(* Logix 5000 project; controller TEC_81 vendor 1 type 14 code 148 rev 36.11; software revision 36.00; part 5 of 5 *)
(* tags used below, declared in another part *)
   Lasers_OK : BOOL;   // Laser Scanner Close Loop Indicator
   LS_1 : DCI_STOP;   // Status of Laser Scanner 1
   LS_1_Status : BOOL;   // General status of inputs
   LS_2 : DCI_STOP;   // Status of Laser Scanner 2
   LS_2_Status : BOOL;   // General status of inputs
   Mat_1_Status : BOOL;   // General status of inputs
   ONS_Laser_1 : BOOL;   // One time execution for reset
   ONS_Laser_2 : BOOL;   // One time execution for reset
   Output_Enable_Laser_1 : BOOL;   // General status of Laser 1
   Output_Enable_Laser_2 : BOOL;   // General status of Laser 2
   Safety_Close_Loop_ok : BOOL;   // General Safety Indicator
   Safety_Mat_ok : BOOL;   // Safety Mat Close Loop Indicator
   Safety_Reset_General : BOOL;   // Unified General Reset
   AbrirInterlock_conveyor_Safety : BOOL;   // Mapped green button for interlock 2 opening
   AbrirInterlock_Principal_Safety : BOOL;   // Mapped green button for interlock 1 opening
   EStops_OK : BOOL;   // E-Stop Close Loop Indicator
   Interlocks_Ok : BOOL;   // Interlocks Close Loop Indicator
   LigthCurtain_ok : BOOL;   // Light Curtains Close Loop Indicator
   MC_1_Interlock : DCI_STOP;   // Status of Interlock 1
   MC_1_Interlock_Status : BOOL;   // General status of inputs
   MC_1_LigthCurtain : DCI_STOP;   // Status of Light Curtain 1
   MC_1_LigthCurtain_Status : BOOL;   // General status of inputs
   MC_2_Interlock : DCI_STOP;   // Status of Interlock 2
   MC_2_Interlock_Status : BOOL;   // General status of inputs
   MC_2_LightCurtain_Status : BOOL;   // General status of inputs
   MC_2_LigthCurtain : DCI_STOP;   // Status of Light Curtain 2
   Ons : INT;
   Operation_Mode : BOOL;   // Operation Mode for HMI (1) Manual (0) Automatico
   Reset_Almacen_1_Sfty : BOOL;
   Reset_Almacen_2_Sfty : BOOL;
   Reset_Principal_Sfty : BOOL;
   Reset_Salida_1_Sfty : BOOL;
   SafetyReset_almacen_1 : BOOL;   // Reset status Almacen 1
   SafetyReset_almacen_2 : BOOL;   // Reset status Almacen 2
   SafetyReset_Principal : BOOL;   // Reset status salida principal
   SafetyReset_Salida_1 : BOOL;   // Reset status Salida 1
   Storage_2 : BOOL;
   Storage_3 : BOOL;
   Storage_4 : BOOL;
   Storage_5 : BOOL;
(* SafetyProgram, continued *)

ROUTINE Interlocks   (* ladder *)
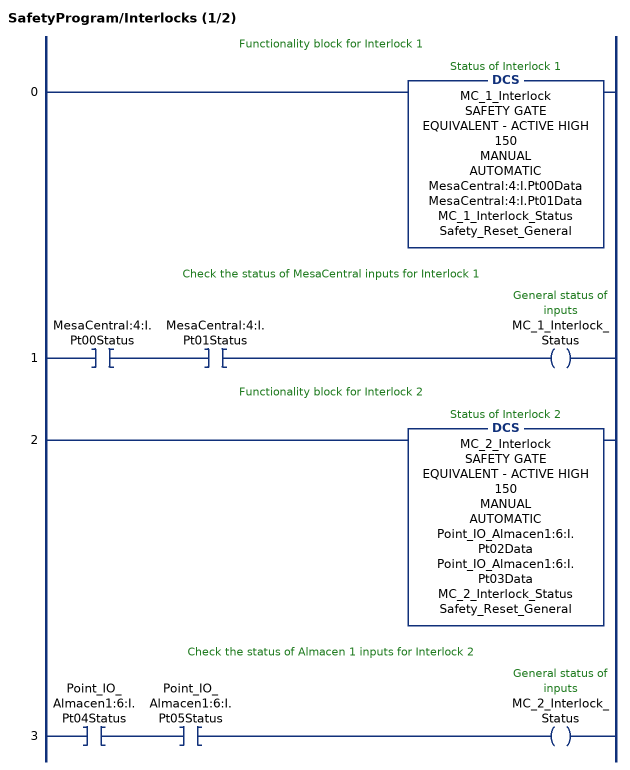
   // Functionality block for Interlock 1
   0: DCS(MC_1_Interlock,SAFETY GATE,EQUIVALENT - ACTIVE HIGH,150,MANUAL,AUTOMATIC,MesaCentral:4:I.Pt00Data,MesaCentral:4:I.Pt01Data,MC_1_Interlock_Status,Safety_Reset_General);
   // Check the status of MesaCentral inputs for Interlock 1
   1: XIC(MesaCentral:4:I.Pt00Status)XIC(MesaCentral:4:I.Pt01Status)OTE(MC_1_Interlock_Status);
   // Functionality block for Interlock 2
   2: DCS(MC_2_Interlock,SAFETY GATE,EQUIVALENT - ACTIVE HIGH,150,MANUAL,AUTOMATIC,Point_IO_Almacen1:6:I.Pt02Data,Point_IO_Almacen1:6:I.Pt03Data,MC_2_Interlock_Status,Safety_Reset_General);
   // Check the status of Almacen 1 inputs for Interlock 2
   3: XIC(Point_IO_Almacen1:6:I.Pt04Status)XIC(Point_IO_Almacen1:6:I.Pt05Status)OTE(MC_2_Interlock_Status);
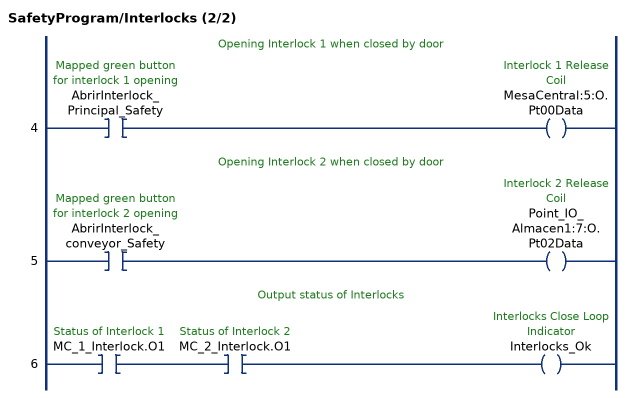
   // Opening Interlock 1 when closed by door
   4: XIC(AbrirInterlock_Principal_Safety)OTE(MesaCentral:5:O.Pt00Data);
   // Opening Interlock 2 when closed by door
   5: XIC(AbrirInterlock_conveyor_Safety)OTE(Point_IO_Almacen1:7:O.Pt02Data);
   // Output status of Interlocks
   6: XIC(MC_1_Interlock.O1)XIC(MC_2_Interlock.O1)OTE(Interlocks_Ok);
END_ROUTINE

ROUTINE Laser_Scanner   (* ladder *)
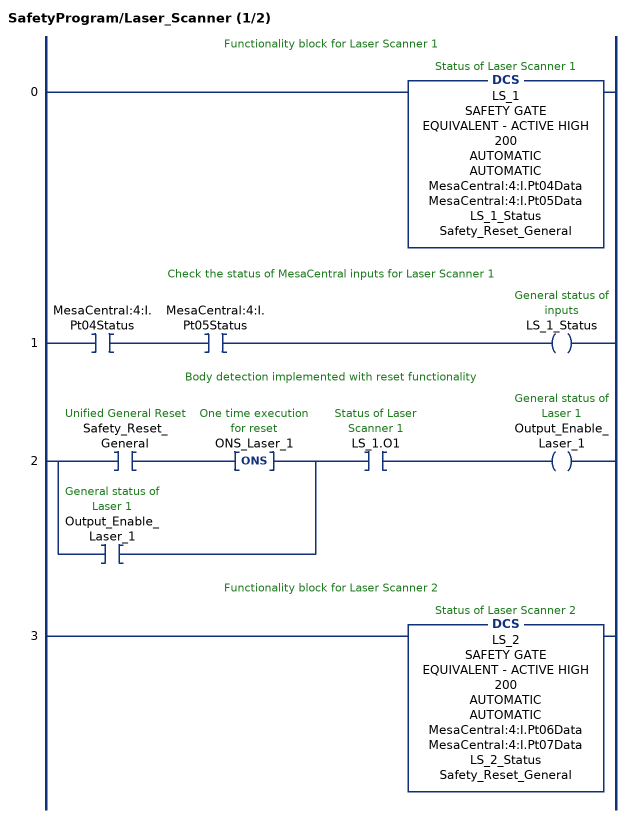
   // Functionality block for Laser Scanner 1
   0: DCS(LS_1,SAFETY GATE,EQUIVALENT - ACTIVE HIGH,200,AUTOMATIC,AUTOMATIC,MesaCentral:4:I.Pt04Data,MesaCentral:4:I.Pt05Data,LS_1_Status,Safety_Reset_General);
   // Check the status of MesaCentral inputs for Laser Scanner 1
   1: XIC(MesaCentral:4:I.Pt04Status)XIC(MesaCentral:4:I.Pt05Status)OTE(LS_1_Status);
   // Body detection implemented with reset functionality
   2: [XIC(Safety_Reset_General) ONS(ONS_Laser_1) ,XIC(Output_Enable_Laser_1) ]XIC(LS_1.O1)OTE(Output_Enable_Laser_1);
   // Functionality block for Laser Scanner 2
   3: DCS(LS_2,SAFETY GATE,EQUIVALENT - ACTIVE HIGH,200,AUTOMATIC,AUTOMATIC,MesaCentral:4:I.Pt06Data,MesaCentral:4:I.Pt07Data,LS_2_Status,Safety_Reset_General);
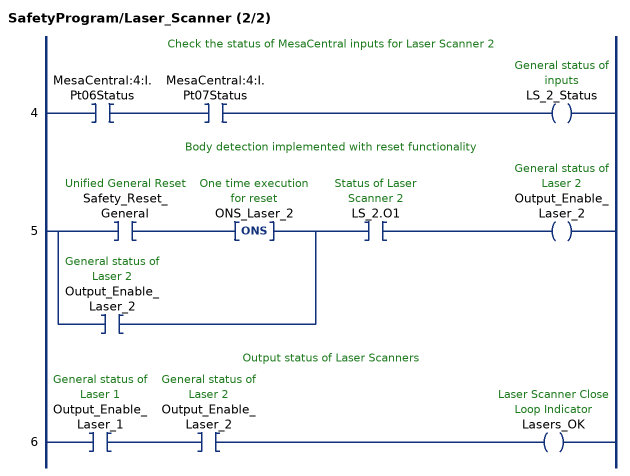
   // Check the status of MesaCentral inputs for Laser Scanner 2
   4: XIC(MesaCentral:4:I.Pt06Status)XIC(MesaCentral:4:I.Pt07Status)OTE(LS_2_Status);
   // Body detection implemented with reset functionality
   5: [XIC(Safety_Reset_General) ONS(ONS_Laser_2) ,XIC(Output_Enable_Laser_2) ]XIC(LS_2.O1)OTE(Output_Enable_Laser_2);
   // Output status of Laser Scanners
   6: XIC(Output_Enable_Laser_1)XIC(Output_Enable_Laser_2)OTE(Lasers_OK);
END_ROUTINE

ROUTINE LigthCurrtains   (* ladder *)
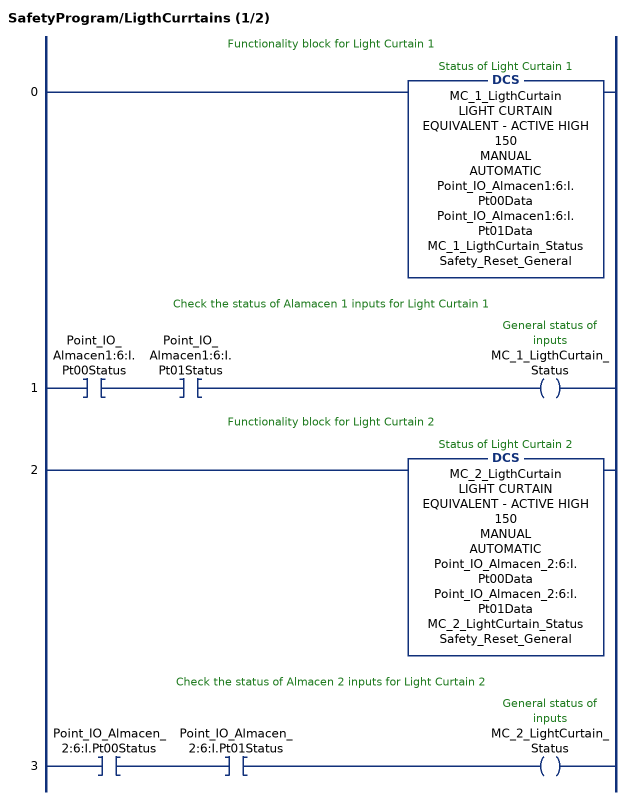
   // Functionality block for Light Curtain 1
   0: DCS(MC_1_LigthCurtain,LIGHT CURTAIN,EQUIVALENT - ACTIVE HIGH,150,MANUAL,AUTOMATIC,Point_IO_Almacen1:6:I.Pt00Data,Point_IO_Almacen1:6:I.Pt01Data,MC_1_LigthCurtain_Status,Safety_Reset_General);
   // Check the status of Alamacen 1 inputs for Light Curtain 1
   1: XIC(Point_IO_Almacen1:6:I.Pt00Status)XIC(Point_IO_Almacen1:6:I.Pt01Status)OTE(MC_1_LigthCurtain_Status);
   // Functionality block for Light Curtain 2
   2: DCS(MC_2_LigthCurtain,LIGHT CURTAIN,EQUIVALENT - ACTIVE HIGH,150,MANUAL,AUTOMATIC,Point_IO_Almacen_2:6:I.Pt00Data,Point_IO_Almacen_2:6:I.Pt01Data,MC_2_LightCurtain_Status,Safety_Reset_General);
   // Check the status of Almacen 2 inputs for Light Curtain 2
   3: XIC(Point_IO_Almacen_2:6:I.Pt00Status)XIC(Point_IO_Almacen_2:6:I.Pt01Status)OTE(MC_2_LightCurtain_Status);
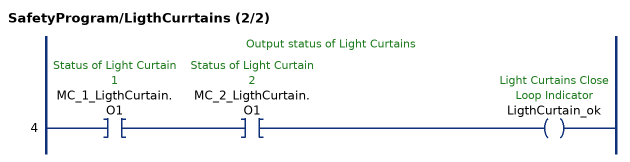
   // Output status of Light Curtains
   4: XIC(MC_1_LigthCurtain.O1)XIC(MC_2_LigthCurtain.O1)OTE(LigthCurtain_ok);
END_ROUTINE

ROUTINE MainRoutine   (* ladder *)
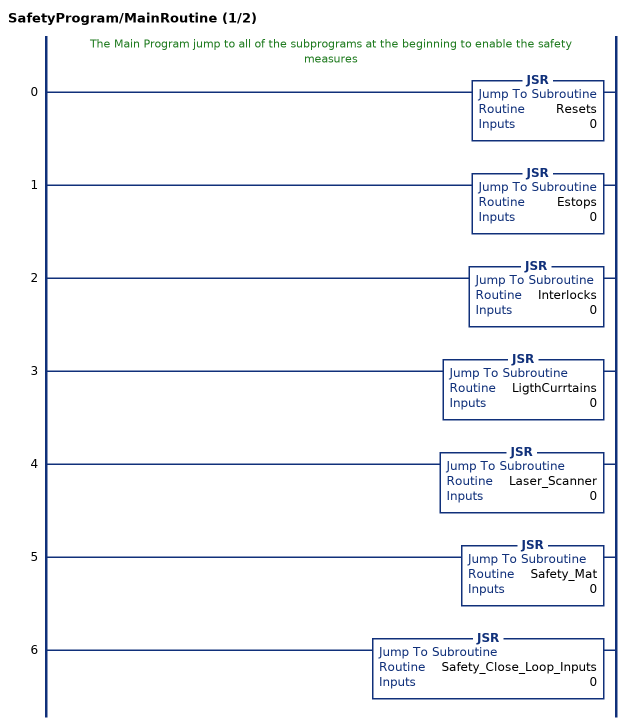
   // The Main Program jump to all of the subprograms at the beginning to enable the safety measures
   0: JSR(Resets,0);
   1: JSR(Estops,0);
   2: JSR(Interlocks,0);
   3: JSR(LigthCurrtains,0);
   4: JSR(Laser_Scanner,0);
   5: JSR(Safety_Mat,0);
   6: JSR(Safety_Close_Loop_Inputs,0);
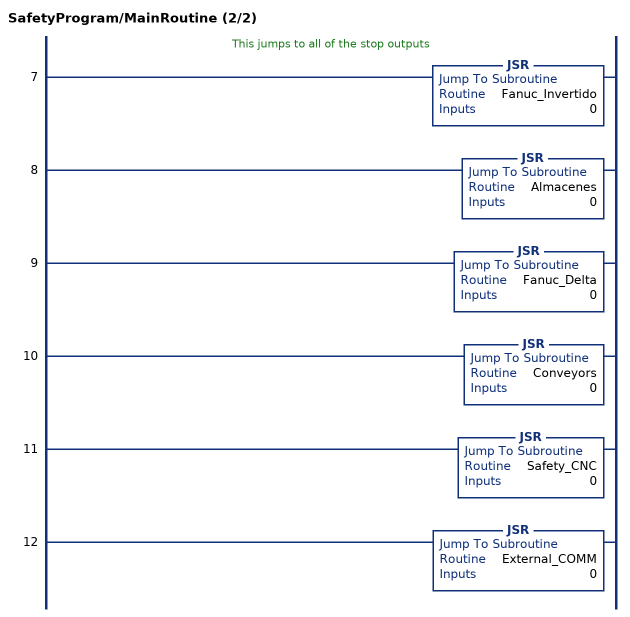
   // This jumps to all of the stop outputs
   7: JSR(Fanuc_Invertido,0);
   8: JSR(Almacenes,0);
   9: JSR(Fanuc_Delta,0);
   10: JSR(Conveyors,0);
   11: JSR(Safety_CNC,0);
   12: JSR(External_COMM,0);
END_ROUTINE

ROUTINE Resets   (* ladder *)
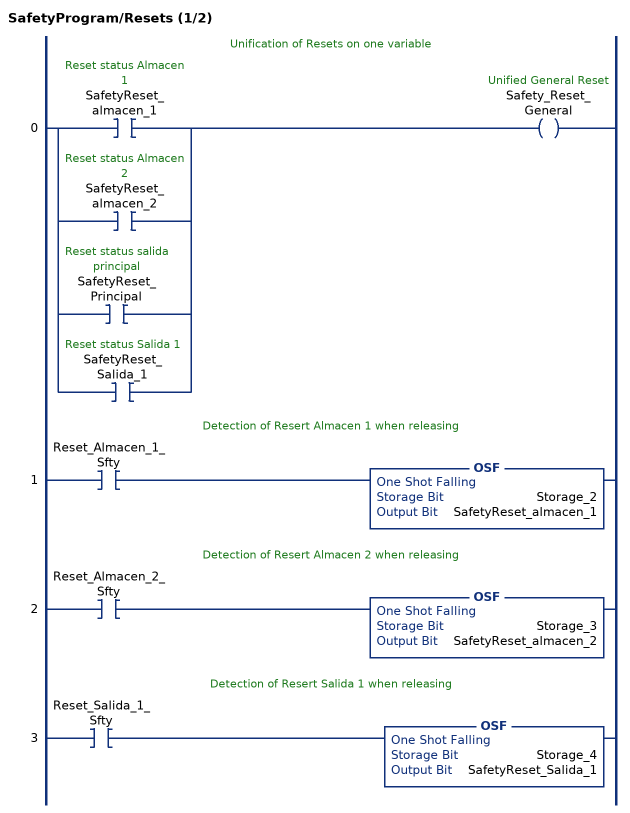
   // Unification of Resets on one variable
   0: [XIC(SafetyReset_almacen_1) ,XIC(SafetyReset_almacen_2) ,XIC(SafetyReset_Principal) ,XIC(SafetyReset_Salida_1) ]OTE(Safety_Reset_General);
   // Detection of Resert Almacen 1 when releasing
   1: XIC(Reset_Almacen_1_Sfty)OSF(Storage_2,SafetyReset_almacen_1);
   // Detection of Resert Almacen 2 when releasing
   2: XIC(Reset_Almacen_2_Sfty)OSF(Storage_3,SafetyReset_almacen_2);
   // Detection of Resert Salida 1 when releasing
   3: XIC(Reset_Salida_1_Sfty)OSF(Storage_4,SafetyReset_Salida_1);
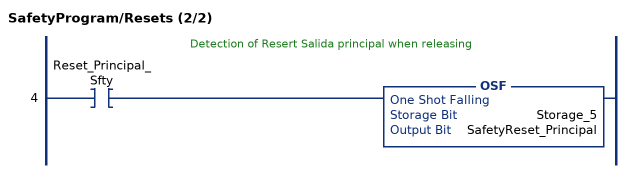
   // Detection of Resert Salida principal when releasing
   4: XIC(Reset_Principal_Sfty)OSF(Storage_5,SafetyReset_Principal);
END_ROUTINE

ROUTINE Safety_Close_Loop_Inputs   (* ladder *)
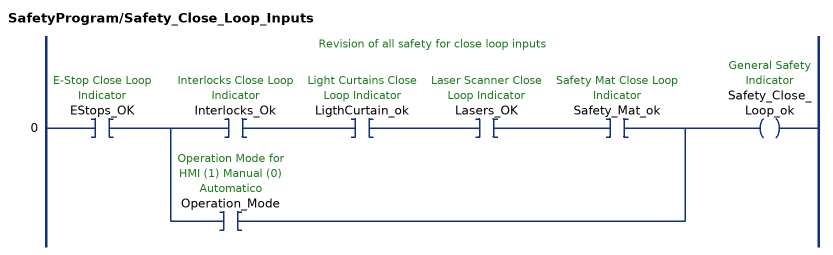
   // Revision of all safety for close loop inputs
   0: XIC(EStops_OK)[XIC(Interlocks_Ok) XIC(LigthCurtain_ok) XIC(Lasers_OK) XIC(Safety_Mat_ok) ,XIC(Operation_Mode) ]OTE(Safety_Close_Loop_ok);
END_ROUTINE

ROUTINE Safety_CNC   (* ladder *)
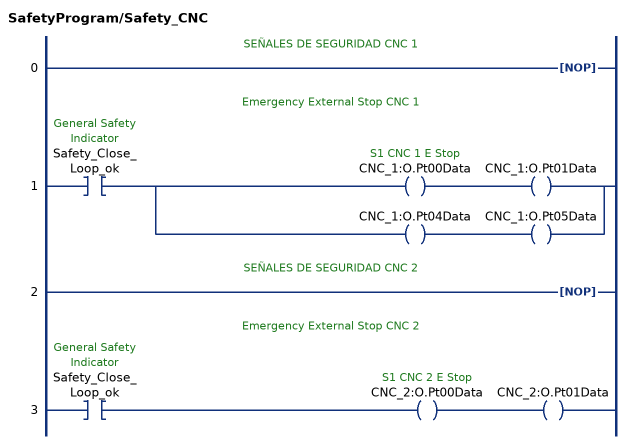
   // SEÑALES DE SEGURIDAD CNC 1
   0: NOP();
   // Emergency External Stop CNC 1
   1: XIC(Safety_Close_Loop_ok)[OTE(CNC_1:O.Pt00Data) OTE(CNC_1:O.Pt01Data) ,OTE(CNC_1:O.Pt04Data) OTE(CNC_1:O.Pt05Data) ];
   // SEÑALES DE SEGURIDAD CNC 2
   2: NOP();
   // Emergency External Stop CNC 2
   3: XIC(Safety_Close_Loop_ok)OTE(CNC_2:O.Pt00Data)OTE(CNC_2:O.Pt01Data);
END_ROUTINE

ROUTINE Safety_Mat   (* ladder *)
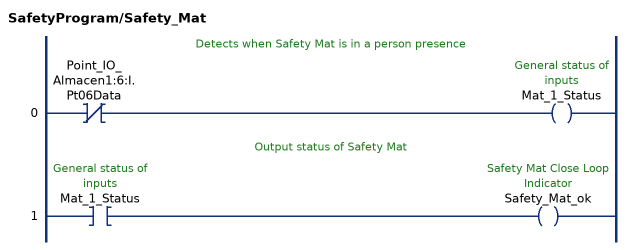
   // Detects when Safety Mat is in a person presence
   0: XIO(Point_IO_Almacen1:6:I.Pt06Data)OTE(Mat_1_Status);
   // Output status of Safety Mat
   1: XIC(Mat_1_Status)OTE(Safety_Mat_ok);
END_ROUTINE
END_PROGRAM
